ADAPTER AGripper
  (* Standard: 61499-1 *)
  (* Version 1.0, 2018-07-09, az *)
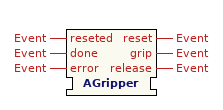
  EVENT_INPUT
    reseted; (* Reseting of cylinder performed succesfully *)
    done; (* action performed succesfully *)
    error; (* an error occured during one of the movements *)
  END_EVENT
  EVENT_OUTPUT
    reset; (* put the cylinder into the inital position (default is home) *)
    grip; (* perform grip movement *)
    release; (* perform release movement *)
  END_EVENT
  SERVICE SOCKET/PLUG
    SEQUENCE request_confirm
      SOCKET.REQ(REQD) -> PLUG.REQ(REQD);
      PLUG.CNF(CNFD) -> SOCKET.CNF(CNFD);
    END_SEQUENCE
    SEQUENCE indication_response
      PLUG.IND(INDD) -> SOCKET.IND(INDD);
      SOCKET.RSP(RSPD) -> PLUG.RSP(RSPD);
    END_SEQUENCE
  END_SERVICE
END_ADAPTER
